INTERFACE I_KNX_DPT_Interpreter

METHOD M_InterpretAs2Bit : ST_KNX_DPT_B2
VAR_IN_OUT
	stInData		: ARRAY[*] OF BYTE;
END_VAR
END_METHOD

METHOD M_InterpretAsBool : BOOL
VAR_IN_OUT
	stInData		: ARRAY[*] OF BYTE;
END_VAR
END_METHOD

METHOD M_InterpretAsDimming : ST_KNX_DPT_ControlDimming
VAR_IN_OUT
	stInData		: ARRAY[*] OF BYTE;
END_VAR
END_METHOD

METHOD M_InterpretAsFloat16 : REAL
VAR_IN_OUT
	stInData		: ARRAY[*] OF BYTE;
END_VAR
END_METHOD

METHOD M_InterpretAsFloat32 : Real
VAR_INPUT
	stInData		: ARRAY[*] OF BYTE;
END_VAR
END_METHOD

METHOD M_InterpretAsINT16 : INT
VAR_IN_OUT
	stInData		: ARRAY[*] OF BYTE;
END_VAR
END_METHOD

METHOD M_InterpretAsINT32 : DINT
VAR_IN_OUT
	stInData		: ARRAY[*] OF BYTE;
END_VAR
END_METHOD

METHOD M_InterpretAsUINT16 : UINT
VAR_IN_OUT
	stInData		: ARRAY[*] OF BYTE;
END_VAR
END_METHOD

METHOD M_InterpretAsUINT32 : UDINT
VAR_IN_OUT
	stInData		: ARRAY[*] OF BYTE;
END_VAR
END_METHOD

METHOD M_InterpretAsUINT8 : BYTE
VAR_IN_OUT
	stInData		: ARRAY[*] OF BYTE;
END_VAR
END_METHOD

METHOD M_InterpretNewMessage : BOOL
VAR_INPUT
	stInData		: BOOL;
END_VAR
END_METHOD

END_INTERFACE

(* stored: Version 1.1.0.1
   Itf I_KNX_DPT_Interpreter: Id {9fb5efa2-43ca-4003-b7af-c2a145e83867}
   Method M_InterpretAs2Bit: Id {66091294-439d-4614-a3f3-24b1c57c3dd4}
   Method M_InterpretAsBool: Id {59cb60ce-9f4b-4da2-ab52-ff9a107f3b72}
   Method M_InterpretAsDimming: Id {7d273548-9943-40e1-9435-3b4660e712af}
   Method M_InterpretAsFloat16: Id {ea166d7f-9d93-4e3b-ad30-38ed3450886a}
   Method M_InterpretAsFloat32: Id {ec4095e0-de89-4da6-8872-91cb0fa9fd48}
   Method M_InterpretAsINT16: Id {ddfdcc34-3a09-41e1-a4d1-3a9db6d7f146}
   Method M_InterpretAsINT32: Id {d212f266-b1d7-4635-8da3-d59af9c13f81}
   Method M_InterpretAsUINT16: Id {33faba98-2ea6-4e4a-ae36-dfb6783a41f1}
   Method M_InterpretAsUINT32: Id {cf65e3be-abb2-4023-85dd-3439bf54739c}
   Method M_InterpretAsUINT8: Id {c3f4480a-1ee3-4276-8307-4f619bec62d2}
   Method M_InterpretNewMessage: Id {0bed79c4-83e7-459c-8517-2c6a14e1e1b8} *)
